PROGRAM P00_OEE
VAR
	//Czasy cyklu 
	fbOEECycleTimes							: FB_OEECycleTimes;
	//Powody odrzuceń           			
	fbOEERejectionReason1					: FB_OEERejectionReason;
	fbOEERejectionReason2					: FB_OEERejectionReason;
	//Przezbrajanie             			
	fbMachinePartsChangeover				: FB_InputFilter;
	
	rtChangeover							: R_TRIG;
	rtfbOEERejectionReason2bDone			: R_TRIG;
	
	sOEERejectionReason1Temp				: STRING;
	sOEERejectionReason2Temp				: STRING;
	
	ifbOEERejectionReason2bAddReasonCount	: INT;
	ifbOEERejectionReason1bAddReasonCount	: INT;
	irtfbOEERejectionReason2bDoneCount		: INT;
	rtfbOEERejectionReason1bDone: R_TRIG;
	irtfbOEERejectionReason1bDoneCount: INT;
	rtORRAdd1sec: R_TRIG;
	tofIbBottleInFormCheckBottleSensor : TOF;

	fbOEERaportLog							: FB_SaveLineToFile;	
	rtOEERaportLogAddLine					: R_TRIG;
	wOEERaportMinuteTemp					: WORD;

	fbOEERaportRejectionLog					: FB_SaveLineToFile;	
	sOEEDateAndTime							: STRING;
	sOEEFileDateAndTime						: STRING;
	sOEEFRejectionLine						: STRING;
	rtOEERaportChooseRecipe					: R_TRIG;	
	bOEETest1								: BOOL;
	tonbOEEGenRaport						: TON;
	sOEEActiveErrorIDs						: STRING;
END_VAR

aCycleTimes();
aRejectionReason();
aMachinePartsChangeover();
aOEETime();
aOEERaport();
aOEEPackMLSuspendedReason();

ACTION aCycleTimes:


tMachineCycleTime;

P02_Dispencers.fbDispencersDragRightStation.tCycleTime;
P02_Dispencers.fbDispencersDragLeftStation.tCycleTime;

P02_Dispencers.fbDispencer1.tCycleTime;
P02_Dispencers.fbDispencer2.tCycleTime;
P02_Dispencers.fbDispencer3.tCycleTime;
P02_Dispencers.fbDispencer4.tCycleTime;
P02_Dispencers.fbDispencerGatesStation.tCycleTime;
P02_Dispencers.fbDispencersCatch1Station.tCycleTime;
P02_Dispencers.fbDispencersCatch2Station.tCycleTime;
P02_Dispencers.fbDispencersCatch3Station.tCycleTime;
P02_Dispencers.fbDispencersCatch4Station.tCycleTime;


P05_Weight.fbWeight1.tCycleTime;
P05_Weight.fbWeight2.tCycleTime;
P05_Weight.fbWeight3.tCycleTime;
P05_Weight.fbWeight4.tCycleTime;


P09_CapPuttedCheck.fbCapPuttedCheck.tCycleTime;

P10_GripperScrewer.fb2GripperScrewer1.tCycleTime;
P10_GripperScrewer.fb2GripperScrewer2.tCycleTime;
P10_GripperScrewer.fbGripperScrewer1CatchStation.tCycleTime;
P10_GripperScrewer.fbGripperScrewer2CatchStation.tCycleTime;

P01_Gates.fbGateBeforeDispencers.tCycleTime;
P13_BottleTransfer.fbBottleTransfer.tCycleTime;




fbOEECycleTimes(
	bEnable:= TRUE, 
	bReset:= FALSE, 
	tStation1CT:= tMachineCycleTime, 
	bStation1En:= TRUE, 
	sStation1Name:= 'M', 
	tStation2CT:= P01_BottleFeeder.fbBottleFeeder.tCycleTime, 
	bStation2En:= P01_BottleFeeder.fbBottleFeeder.bEnable, 
	sStation2Name:= 'SORB', 
	tStation3CT:= P02_Dispencers.fbDispencersDragRightStation.tCycleTime , 
	bStation3En:= P02_Dispencers.fbDispencersDragRightStation.bEnable, 
	sStation3Name:= 'PFDP', 
	tStation4CT:= P02_Dispencers.fbDispencersDragLeftStation.tCycleTime, 
	bStation4En:= P02_Dispencers.fbDispencersDragLeftStation.bEnable, 
	sStation4Name:= 'PFDL', 
	tStation5CT:= P02_Dispencers.fbDispencer1.tCycleTime, 
	bStation5En:= P02_Dispencers.fbDispencer1.bEnable, 
	sStation5Name:= 'D1', 
	tStation6CT:= P02_Dispencers.fbDispencer2.tCycleTime, 
	bStation6En:= P02_Dispencers.fbDispencer2.bEnable,
	sStation6Name:= 'D2', 
	tStation7CT:= P02_Dispencers.fbDispencer3.tCycleTime, 
	bStation7En:= P02_Dispencers.fbDispencer3.bEnable, 
	sStation7Name:= 'D3', 
	tStation8CT:= P02_Dispencers.fbDispencer4.tCycleTime, 
	bStation8En:= P02_Dispencers.fbDispencer4.bEnable, 
	sStation8Name:= 'D4', 
	tStation9CT:= P02_Dispencers.fbDispencersCatch1Station.tCycleTime,
	bStation9En:= P02_Dispencers.fbDispencersCatch1Station.bEnable, 
	sStation9Name:= 'CHD1', 
	tStation10CT:= P02_Dispencers.fbDispencersCatch2Station.tCycleTime, 
	bStation10En:= P02_Dispencers.fbDispencersCatch2Station.bEnable, 
	sStation10Name:= 'CHD2', 
	tStation11CT:= P02_Dispencers.fbDispencersCatch3Station.tCycleTime, 
	bStation11En:= P02_Dispencers.fbDispencersCatch3Station.bEnable,
	sStation11Name:= 'CHD3', 
	tStation12CT:=  P02_Dispencers.fbDispencersCatch4Station.tCycleTime, 
	bStation12En:= P02_Dispencers.fbDispencersCatch4Station.bEnable, 
	sStation12Name:=  'CHD4', 
	tStation13CT:= P05_Weight.fbWeightStation.tCycleTime,
	bStation13En:= P05_Weight.fbWeightStation.bEnable, 
	sStation13Name:= 'PW',
	tStation14CT:= P05_Weight.fbWeightStation2Phase.tCycleTime,
	bStation14En:= P05_Weight.fbWeightStation2Phase.bEnable, 
	sStation14Name:= 'PW',	
	tStation15CT:= P05_Weight.fbWeight1.tCycleTime, 
	bStation15En:= P05_Weight.fbWeight1.bEnable, 
	sStation15Name:= 'W1', 
	tStation16CT:= P05_Weight.fbWeight2.tCycleTime, 
	bStation16En:= P05_Weight.fbWeight2.bEnable, 
	sStation16Name:= 'W2',  
	tStation17CT:= P05_Weight.fbWeight3.tCycleTime, 
	bStation17En:= P05_Weight.fbWeight3.bEnable, 
	sStation17Name:= 'W3',  
	tStation18CT:= P05_Weight.fbWeight4.tCycleTime, 
	bStation18En:= P05_Weight.fbWeight4.bEnable, 
	sStation18Name:= 'W4',  
	tStation19CT:= P05_Weight.fbWeight5.tCycleTime,  
	bStation19En:= P05_Weight.fbWeight5.bEnable,
	sStation19Name:= 'W5',
	tStation20CT:= P05_Weight.fbWeight6.tCycleTime,  
	bStation20En:= P05_Weight.fbWeight6.bEnable, 
	sStation20Name:= 'W6',  
	tStation21CT:= P10_GripperScrewer.fbGripperScrewersDragStation.tCycleTime, 
	bStation21En:= P10_GripperScrewer.fbGripperScrewersDragStation.bEnable,
	sStation21Name:= 'PFDZ',
	tStation22CT:= P10_GripperScrewer.fb2GripperScrewer1.tCycleTime, 
	bStation22En:= P10_GripperScrewer.fb2GripperScrewer1.bEnable1,
	sStation22Name:= 'ZS1',
	tStation23CT:= P10_GripperScrewer.fb2GripperScrewer2.tCycleTime, 
	bStation23En:= P10_GripperScrewer.fb2GripperScrewer2.bEnable2,
	sStation23Name:= 'ZS2',
	tStation24CT:= P10_GripperScrewer.fbGripperScrewersDragStation.tCycleTime, 
	bStation24En:= P10_GripperScrewer.fbGripperScrewersDragStation.bEnable,
	sStation24Name:= 'PFZ',
	tStation25CT:= P10_GripperScrewer.fbGripperScrewer1CatchStation.tCycleTime, 
	bStation25En:= P10_GripperScrewer.fbGripperScrewer1CatchStation.bEnable,
	sStation25Name:= 'CHZS1',
	tStation26CT:= P10_GripperScrewer.fbGripperScrewer2CatchStation.tCycleTime, 
	bStation26En:= P10_GripperScrewer.fbGripperScrewer2CatchStation.bEnable,
	sStation26Name:= 'CHZS2',
	tStation27CT:= P11_CapCorrectCheck.fbCapCorrectCheck.tCycleTime, 
	bStation27En:= P11_CapCorrectCheck.fbCapCorrectCheck.bEnable,
	sStation27Name:= 'SZA',
	tStation28CT:= P13_BottleTransfer.fbBottleTransfer.tCycleTime, 
	bStation28En:= P13_BottleTransfer.fbBottleTransfer.bEnable,
	sStation28Name:= 'R',  
	tStation29CT:= P01_Gates.fbGateBeforeDispencers.tCycleTime, 
	bStation29En:= P01_Gates.fbGateBeforeDispencers.bEnable, 
	sStation29Name:= 'SZD', 
	tStation20CT:= P01_Gates.fbGateRobot.tCycleTime, 
	bStation30En:= P01_Gates.fbGateRobot.bEnable, 
	sStation30Name:= 'SZR', 

	
	
	AsCycleTimes=> VIS.AsOEECycleTimes,
	
	
	
	);
END_ACTION

ACTION aMachinePartsChangeover:

VIS.bMachinePartsChangeOver	;						// Włączone przezbrajanie (ustawić z wizki)
VIS.iMachinePartsChangeOver	;						// Stan przezbrajania (0-ruch,1-pozycja gorna,-1-pozycja dolna) 
VIS.bBottleSorterDisable	;						// Wyłączenie sortera butelek
VIS.bCapSorterDisable		;						// Wyłączenie sortera nasadek


//Sygnał z wizki
VIS.bMachinePartsChangeover;
//Filtrowanie sygnału, przeciw lagom z wizualizacji lub ciągłym klikaniem
fbMachinePartsChangeover(bIn:=VIS.bMachinePartsChangeover,tFilterTimeOn:=T#3S,tFilterTimeOff:=T#3S,bOUT=>bChangeover);
//Przefiltrowany
bChangeover;

VIS.iMachinePartsChangeOver;
// Trzeba dodać, albo wyłączona stacja!
//Przezbrajanie - okienko 


IF bChangeover THEN
	VIS.bBottleSorterHold	:= TRUE;	
	VIS.bCapSorterHold		:= TRUE;	
	//VIS.bTank1SupplyPumpEnableShow:=FALSE;
	//VIS.bTank2SupplyPumpEnableShow:=FALSE;
ELSE
	//VIS.bBottleSorterHold	:= FALSE;	
	VIS.bCapSorterHold		:= FALSE;			
END_IF

IF 
 (P02_Dispencers.fbDispencersCatch1Station.eState = E_Station.ePreparingToDisable 			OR P02_Dispencers.fbDispencersCatch1Station.eState = E_Station.eHoming 				OR (NOT bDispencer1Enable AND NOT bDispencer3Enable)) 																			AND
 (P09_CapPuttedCheck.fbCapPuttedCheck.eState = E_Station.ePreparingToDisable				OR P09_CapPuttedCheck.fbCapPuttedCheck.eState = E_Station.eHoming				 	OR NOT bCapPuttedCheckEnable) 									AND
 (P10_GripperScrewer.fb2GripperScrewer1.eState = E_Station.ePreparingToDisable				OR P10_GripperScrewer.fb2GripperScrewer1.eState = E_Station.eHoming  				OR NOT bGripperScrewer1Enable) 									AND
 (P10_GripperScrewer.fb2GripperScrewer2.eState = E_Station.ePreparingToDisable				OR P10_GripperScrewer.fb2GripperScrewer2.eState = E_Station.eHoming  				OR NOT bGripperScrewer2Enable)									AND
 (P10_GripperScrewer.fbGripperScrewer1CatchStation.eState = E_Station.ePreparingToDisable 	OR P10_GripperScrewer.fbGripperScrewer1CatchStation.eState = E_Station.eHoming		OR NOT bGripperScrewer1Enable) 									AND
 (P10_GripperScrewer.fbGripperScrewer2CatchStation.eState = E_Station.ePreparingToDisable 	OR P10_GripperScrewer.fbGripperScrewer2CatchStation.eState = E_Station.eHoming 		OR NOT bGripperScrewer2Enable) 									AND
 (P11_CapCorrectCheck.fbCapCorrectCheck.eState = E_Station.ePreparingToDisable 				OR P11_CapCorrectCheck.fbCapCorrectCheck.eState = E_Station.eHoming					OR NOT bCapCorrectCheckEnable)
THEN
    VIS.iMachinePartsChangeOver := 0; //ruch
ELSIF
  (P02_Dispencers.fbDispencersCatch1Station.eState = E_Station.eDisabled			OR P02_Dispencers.fbDispencersCatch1Station.eState = E_Station.eManualMovement 			OR (NOT bDispencer1Enable AND NOT bDispencer3Enable) ) 											AND
 (P09_CapPuttedCheck.fbCapPuttedCheck.eState = E_Station.eDisabled				 	OR NOT bCapPuttedCheckEnable) 										AND
 (P10_GripperScrewer.fb2GripperScrewer1.eState = E_Station.eDisabled  				OR NOT bGripperScrewer1Enable)										AND
 (P10_GripperScrewer.fb2GripperScrewer2.eState = E_Station.eDisabled  				OR	NOT bGripperScrewer2Enable)										AND
 (P10_GripperScrewer.fbGripperScrewer1CatchStation.eState = E_Station.eDisabled 	OR NOT bGripperScrewer1Enable) 										AND
 (P10_GripperScrewer.fbGripperScrewer2CatchStation.eState = E_Station.eDisabled 	OR NOT bGripperScrewer2Enable) 										AND
 (P11_CapCorrectCheck.fbCapCorrectCheck.eState = E_Station.eDisabled 				OR NOT bCapCorrectCheckEnable)
THEN
    VIS.iMachinePartsChangeOver := 1; //1 pozycja gorna
ELSIF 
  (P02_Dispencers.fbDispencersCatch1Station.eState = E_Station.eReady 		OR P02_Dispencers.fbDispencersCatch1Station.eState = E_Station.eManualMovement 				OR (NOT bDispencer1Enable AND NOT bDispencer3Enable)) 												AND
 (P09_CapPuttedCheck.fbCapPuttedCheck.eState = E_Station.eReady				OR P09_CapPuttedCheck.fbCapPuttedCheck.eState = E_Station.eManualMovement			 		OR NOT bCapPuttedCheckEnable) 											AND
 (P10_GripperScrewer.fb2GripperScrewer1.eState = E_Station.eReady  			OR P10_GripperScrewer.fb2GripperScrewer1.eState = E_Station.eManualMovement					OR NOT bGripperScrewer1Enable)											AND
 (P10_GripperScrewer.fb2GripperScrewer2.eState = E_Station.eReady  			OR P10_GripperScrewer.fb2GripperScrewer2.eState = E_Station.eManualMovement					OR NOT bGripperScrewer2Enable) 											AND
 (P10_GripperScrewer.fbGripperScrewer1CatchStation.eState = E_Station.eReady OR P10_GripperScrewer.fbGripperScrewer1CatchStation.eState = E_Station.eManualMovement		OR NOT bGripperScrewer1Enable) 											AND
 (P10_GripperScrewer.fbGripperScrewer2CatchStation.eState = E_Station.eReady OR P10_GripperScrewer.fbGripperScrewer2CatchStation.eState = E_Station.eManualMovement		OR NOT bGripperScrewer2Enable) 											AND
 (P11_CapCorrectCheck.fbCapCorrectCheck.eState = E_Station.eReady 			OR	P11_CapCorrectCheck.fbCapCorrectCheck.eState = E_Station.eManualMovement 				OR NOT bCapCorrectCheckEnable)
THEN
    VIS.iMachinePartsChangeOver := -1; // -1pozycja dolna
END_IF 

//Kasowanie cyklu i liczników
rtChangeover(CLK:=bChangeover,Q=>);
IF rtChangeover.Q THEN
	//bCycleReseting := TRUE;	
	VIS.uiCounterAverageEfficiency:=0;
	VIS.udiCounterShiftBottles:=0;
	VIS.uiCounterInstantEfficiency:=0;
	VIS.uiCounterGoodBottles:=0;
	VIS.uiCounterBadBottles:=0;
END_IF
END_ACTION

ACTION aOEEPackMLSuspendedReason:
(*
Nazwa:			aOEEPackMLSuspendedReason
Wersja:			v0.1 			
Autor:			DP
Urzadzenia:		HMI, 
Konfiguracja:	
Info:
- Wyświetlanie na wykresie powodu zatrzymania lini, czyli w przyszłości przjeścia w stan PackML ->Suspended
Uwagi:

Zmiany:

*)
IF P00_PackML.tonCycleBadBottleConveyorFullSensor.Q THEN //odrzut
	VIS.iOEEPackMLSuspendedReason	:= 1;
ELSIF P16_LabelMachine.tonLabelMachineFullSensorInfo.Q THEN 
	//IF VIS.UPPackMLState=6 AND VIS.EPPackMLState=6 THEN		//etykieciarka
	VIS.iOEEPackMLSuspendedReason	:= 2;
ELSIF	vis.iMachineState = 2 OR vis.iMachineState = 8 OR vis.iMachineState = 9 OR vis.iMachineState = 15 THEN
	VIS.iOEEPackMLSuspendedReason	:= 3;
	//ELSIF VIS.UPPackMLState<>6 AND VIS.EPPackMLState=6 THEN //kartoniarka
	//VIS.iOEEPackMLSuspendedReason	:= 7;
	//ELSIF VIS.UPPackMLState=6 AND VIS.EPPackMLState<>6 THEN //paletyzer
	//VIS.iOEEPackMLSuspendedReason	:= 8;
	//END_IF
//ELSIF VIS.uliWarningOccure.33 THEN  //brak butelek
//	VIS.iOEEPackMLSuspendedReason	:= 3;	
//ELSIF VIS.uliWarningOccure.27 THEN	//brak nakrętek
//	VIS.iOEEPackMLSuspendedReason	:= 4;	
//(*ELSIF NOT P16_LabelMachine.tonLabelMachineFullSensorInfo.Q THEN		
//	IF VIS.UPPackMLState<>6 AND VIS.EPPackMLState=6 THEN			//kartoniarka
//	VIS.iOEEPackMLSuspendedReason	:= 7;
//	ELSIF VIS.UPPackMLState=6 AND VIS.EPPackMLState<>6 THEN			//paletyzer
//	VIS.iOEEPackMLSuspendedReason	:= 8;
//	END_IF*)
ELSE
	VIS.iOEEPackMLSuspendedReason	:= 0;		
END_IF
END_ACTION

ACTION aOEERaport:

//Data dla danych - według opisu
sOEEDateAndTime:= 
Concat(Concat(Concat(Concat(Concat(Concat(Concat(Concat(Concat(Concat(Concat(WORD_TO_STRING(wDay),'.'),WORD_TO_STRING(wMonth)),'.'),WORD_TO_STRING(wYear)),';'),WORD_TO_STRING(wHour)),':'),WORD_TO_STRING(wMinute)),';'),''),'');

//Generowanie raportu z wizki - podpiąć pod wybór receptury?
VIS.bOEEGenRaport;

//Zapisywanie daty wybrania receptury
//rtOEERaportChooseRecipe(CLK:=VIS.bChooseRecipe OR bOEETest1, Q=>);
rtOEERaportChooseRecipe(CLK:=VIS.bOEEGenRaport OR bOEETest1, Q=>);
tonbOEEGenRaport(IN:=VIS.bOEEGenRaport, PT:=T#500MS);
IF rtOEERaportChooseRecipe.Q THEN
	sOEEFileDateAndTime:= 
	Concat(Concat(Concat(Concat(Concat(Concat(Concat(Concat(Concat(Concat(Concat(WORD_TO_STRING(wYear),''),WORD_TO_STRING(wMonth)),''),WORD_TO_STRING(wDay)),''),WORD_TO_STRING(wHour)),''),WORD_TO_STRING(wMinute)),''),''),'');
	bOEETest1	:=	FALSE;
END_IF
IF tonbOEEGenRaport.Q THEN
	VIS.bOEEGenRaport	:= FALSE;
END_IF

//Zapisywanie danych co 1 min
rtOEERaportLogAddLine(CLK:=wMinute <> wOEERaportMinuteTemp, Q=>);	
IF rtOEERaportLogAddLine.Q THEN 
	wOEERaportMinuteTemp := wMinute;
END_IF

//Zapisywanie aktywnych bledow w stringu
IF rtOEERaportLogAddLine.Q THEN
	sOEEActiveErrorIDs := '';
	FOR i:=1 TO 10 DO
		IF VIS.fbAlarms.arrActiveEvents[i].stEventEntry.nEventId <> 0 THEN
			sOEEActiveErrorIDs:=Concat(sOEEActiveErrorIDs,Concat(UDINT_TO_STRING(VIS.fbAlarms.arrActiveEvents[i].stEventEntry.nEventId),';'));	
		END_IF
	END_FOR
	sOEEActiveErrorIDs:= Concat(sOEEActiveErrorIDs,stBottleSorterRead.eError.sStationName);
	sOEEActiveErrorIDs:= Concat(sOEEActiveErrorIDs,stCapSorterRead.eError.sStationName);	
END_IF			
		
//Raport nazwy,liczników itd
fbOEERaportLog(
	bExecute:= rtOEERaportLogAddLine.Q,
	AmsNetId:= , 
	sPath:='C:\Users\Administrator\Desktop\CSVFolder\', 
	sName:= Concat(sOEEFileDateAndTime,	Concat('-',Concat(sRecipeName,'.csv'))), 
	sLine:= 
	
Concat(
	'$R$N',
	Concat(
		sOEEDateAndTime,
		Concat(
				UINT_TO_STRING(VIS.iMachineState),
				Concat(
						';',
							Concat(
									sRecipeName,
									Concat(
											';',
											Concat(
													UDINT_TO_STRING(VIS.udiCounterGlobal),
														Concat(
																';',
																	Concat(
																		UDINT_TO_STRING(VIS.uiCounterBadBottles),
																		Concat(
																			';',
																			Concat(
																					//UDINT_TO_STRING(VIS.udiStationErrorCode),
																					sOEEActiveErrorIDs,
																					';'
																					)	
																				)	
																			)
																)
													)
											)
										)
						)
					)
				)
		)		
	,
	
	bBusy=>, 
	bError=>);

	IF rtOEERaportLogAddLine.Q THEN
		sOEEFRejectionLine := '';
		FOR i:= 0 TO 63 DO
			IF 	VIS.AStBadPackageReason[i].udiID <> 0 THEN
				
				sOEEFRejectionLine := 
					Concat(sOEEFRejectionLine,Concat(UDINT_TO_STRING(VIS.AStBadPackageReason[i].udiID), Concat(';',Concat(WSTRING_TO_STRING(VIS.AStBadPackageReason[i].wsDescription),';'))));
						
			END_IF
		END_FOR
	END_IF

//Raport odrzutów
fbOEERaportRejectionLog(
	bExecute:= rtOEERaportLogAddLine.Q,
	AmsNetId:= , 
	sPath:='C:\Users\Administrator\Desktop\CSVRejectionFolder\', 
	sName:= Concat(sOEEFileDateAndTime,	Concat('-',Concat(sRecipeName,'-Rejection.csv'))), 
	sLine:= Concat('$R$N',sOEEFRejectionLine),
	bBusy=>, 
	bError=>);
END_ACTION

ACTION aOEETime:

VIS.udiCounterShiftBottles;
VIS.udiCounterGlobal;            
VIS.udiCounterGlobalBadBottles;     

VIS.sOEEText1 := Concat(Concat('PRACA: ', UDINT_TO_STRING(udiCounterExecuteTimeTemp/60)),' min');
VIS.sOEEText2 := Concat(Concat('POSTÓJ: ', UDINT_TO_STRING(udiCounterReadyTimeTemp/60)),' min');
VIS.sOEEText3 := Concat(Concat('BŁĄD: ', UDINT_TO_STRING(udiCounterErrorTimeTemp/60)),' min');
tofIbBottleInFormCheckBottleSensor(IN:=MAIN.IbBottleInFormCheckBottleSensor,PT:=T#30S);

VIS.udiCounterExecuteTime	:=	UDINT_TO_UINT(udiCounterExecuteTimeTemp/60);
VIS.udiCounterReadyTime		:=	UDINT_TO_UINT(udiCounterReadyTimeTemp/60);
VIS.udiCounterErrorTime	  	:=	UDINT_TO_UINT(udiCounterErrorTimeTemp/60);
rtORRAdd1sec(CLK:=b2Hz,Q=>);

IF	
	//P00_PackML.fbPMLAuto.ePMLState = Tc3_PackML.E_PMLState.ePMLState_STARTING OR 
	//P00_PackML.fbPMLAuto.ePMLState = Tc3_PackML.E_PMLState.ePMLState_STOPPING OR 
	P00_PackML.fbPMLAuto.ePMLState = Tc3_PackML.E_PMLState.ePMLState_EXECUTE AND
	tofIbBottleInFormCheckBottleSensor.Q AND 
	NOT P16_LabelMachine.tonLabelMachineFullSensorInfo.Q AND
	NOT (P00_PackML.tonCycleBadBottleConveyorFullSensor.Q AND (P00_PackML.iRobotPickCase=110 OR P00_PackML.iRobotPickCase=210))
	THEN

	IF rtORRAdd1sec.Q THEN
		udiCounterExecuteTimeTemp	:=	udiCounterExecuteTimeTemp	+	1;
		
	END_IF
	
ELSIF
	P00_PackML.fbPMLAuto.ePMLState = Tc3_PackML.E_PMLState.ePMLState_STOPPED OR 
	P00_PackML.fbPMLAuto.ePMLState = Tc3_PackML.E_PMLState.ePMLState_ABORTED  
	THEN
	
	IF rtORRAdd1sec.Q THEN
		udiCounterErrorTimeTemp	:=	udiCounterErrorTimeTemp	+	1;
	END_IF	

ELSE
	IF rtORRAdd1sec.Q THEN
		udiCounterReadyTimeTemp	:=	udiCounterReadyTimeTemp	+	1;
	END_IF	
END_IF
END_ACTION

ACTION aRejectionReason:

//może uzależnić też od ilości opakowań do pobrania VIS.nBottleTransferPickOption			:=	1; // 1 butelka
//													VIS.nBottleTransferPlaceOption			:=	2; //Odrzucone butelki 

fbOEERejectionReason1(
                        bEnable				:= TRUE,
                        bReset				:= ,
                        udiGlobalCounter	:= VIS.udiCounterGlobal, //Globalny licznik konfekcji [szt]
                        bAddReason			:= P13_BottleTransfer.fbBottleTransfer.eRunningState>1 AND VIS.nBottleTransferPlaceOption=2, // może dodać dodatkowy warunek?
                        bReason1			:= eRobotPackageState[1].bWeightTooLow 			AND eRobotPackageState[1].bBottlePresent,
                        sReason1Description	:= 'WZM',
                        bReason2			:= eRobotPackageState[1].bWeightTooHigh 		AND eRobotPackageState[1].bBottlePresent,
                        sReason2Description	:= 'WZD',
                        bReason3			:= NOT eRobotPackageState[1].bCapOK 			AND eRobotPackageState[1].bBottlePresent,
                        sReason3Description	:= 'BNPZ',
                        bReason4			:= NOT eRobotPackageState[1].bCapGripperScrewed AND eRobotPackageState[1].bBottlePresent,
                        sReason4Description	:= 'NZZSZ',
                        bReason5			:= NOT eRobotPackageState[1].bCapCorrectCapOn 	AND eRobotPackageState[1].bBottlePresent,
                        sReason5Description	:= 'BNZZ',
                        bReason6			:= eRobotPackageState[1].bCapCorrectNOK 		AND eRobotPackageState[1].bBottlePresent,
                        sReason6Description	:= 'NZZ',
                        bReason7			:=, 
                        sReason7Description	:= ,      
                        sRejectionReason	:= sOEERejectionReason1Temp,
                        );

fbOEERejectionReason2(
                        bEnable				:= TRUE,
                        bReset				:= ,
                        udiGlobalCounter	:= VIS.udiCounterGlobal, //Globalny licznik konfekcji [szt]
                        bAddReason			:= P13_BottleTransfer.fbBottleTransfer.eRunningState>1 AND VIS.nBottleTransferPlaceOption=2,
                        bReason1			:= eRobotPackageState[2].bWeightTooLow 			AND eRobotPackageState[2].bBottlePresent,
                        sReason1Description	:= 'WZM',
                        bReason2			:= eRobotPackageState[2].bWeightTooHigh 		AND eRobotPackageState[2].bBottlePresent,
                        sReason2Description	:= 'WZD',
                        bReason3			:= NOT eRobotPackageState[2].bCapOK 			AND eRobotPackageState[2].bBottlePresent,
                        sReason3Description	:= 'BNPZ',
                        bReason4			:= NOT eRobotPackageState[2].bCapGripperScrewed AND eRobotPackageState[2].bBottlePresent,
                        sReason4Description	:= 'NZZSZ',
                        bReason5			:= NOT eRobotPackageState[2].bCapCorrectCapOn 	AND eRobotPackageState[2].bBottlePresent,
                        sReason5Description	:= 'BNZZ',
                        bReason6			:= eRobotPackageState[2].bCapCorrectNOK 		AND eRobotPackageState[2].bBottlePresent,
                        sReason6Description	:= 'NZZ',
                        bReason7			:= , 
                        sReason7Description	:= ,      
                        sRejectionReason	:= sOEERejectionReason2Temp,
                        );
						
	rtfbOEERejectionReason2bDone(CLK:=fbOEERejectionReason2.bDone,Q=>);
	rtfbOEERejectionReason1bDone(CLK:=fbOEERejectionReason1.bDone,Q=>);
// dodałem na testy! 20.06	
	IF rtfbOEERejectionReason1bDone.Q AND  VIS.nBottleTransferPickOption=1 THEN
		VIS.sOEERejectionReason 			:=sOEERejectionReason1Temp;//	CONCAT(sOEERejectionReason1Temp,';');
		irtfbOEERejectionReason1bDoneCount	:=	irtfbOEERejectionReason1bDoneCount+1;
	END_IF
	
	
	IF rtfbOEERejectionReason2bDone.Q AND  VIS.nBottleTransferPickOption=2 THEN
		VIS.sOEERejectionReason 			:=	CONCAT(CONCAT(sOEERejectionReason1Temp,';'),sOEERejectionReason2Temp);
		irtfbOEERejectionReason2bDoneCount	:=	irtfbOEERejectionReason2bDoneCount+1;
	END_IF
	
    //Przeniesione dodawanie liczników, po to żeby dla wizualizacji i skryptów było łatwiej (kolejnosć odczytu)
    IF bAddGlobalCounter AND (fbOEERejectionReason2.bDone OR fbOEERejectionReason1.bDone )THEN
        VIS.uiCounterBadBottles                	:= VIS.uiCounterBadBottles		+ INT_TO_UINT(P00_PackML.nCounterFormsToLoad);//+ 1;// czy aby na pewno +1 ???
        VIS.udiCounterGlobalBadBottles        	:= VIS.udiCounterGlobalBadBottles	+ INT_TO_UDINT(P00_PackML.nCounterFormsToLoad);
        VIS.udiCounterGlobal                   	:= VIS.udiCounterGlobal			+ INT_TO_UDINT(P00_PackML.nCounterFormsToLoad);
        //VIS.udiCounterShiftBottles            	:= VIS.udiCounterShiftBottles	+ INT_TO_UDINT(P00_PackML.nCounterFormsToLoad);
        bAddGlobalCounter                    	:= FALSE;
    END_IF

    IF fbOEERejectionReason1.bAddReason THEN
       ifbOEERejectionReason1bAddReasonCount:=ifbOEERejectionReason1bAddReasonCount+1;
    END_IF
	
    IF fbOEERejectionReason2.bAddReason THEN
        ifbOEERejectionReason2bAddReasonCount:=ifbOEERejectionReason2bAddReasonCount+1;
     END_IF
END_ACTION

END_PROGRAM

(* stored: Version 1.1.0.1, ProductVersion 3.1.4026.13, FileIdentifier 02689428d8efeed8a78b8ef3a3fdcfe5d09039a9, FileSignature 44daf26e7e7288f74d3f978d1d0214b2b1e5c506aa9bfd24740d0514adf3d7f1fed84f6822c00263c792253789ebda25bdc56938ff42e3c47365d65a564f3c8034953b4d2f9a46ca5952431417d125fd436c812405c40c2e3f75dcfe042a473413b156317058a588511bcd444fc63c9d2a5edcfb8a3e4d1b3007ca2dd304362b15f63a3ef2c8624fa66b21e5af4a2dada87096a7028e7d86cdc7e0a1abc17373387c7f25656e002f963e77048528c9d3ee5a8664849fcff38f7fdd1dda37988d09f68298b31ae6fe10a5b95e2b73eac28d16b4fce65a3f435e9996781ee949c42ed40e4418f2cb3d264bd489d0da85916129245d2c4672d1935a82bfee9b4390
   POU P00_OEE: Id {08c14e30-ec5a-4e4c-b5ac-ce8b40bd55d7}, SpecialFunc None
   Action aCycleTimes: Id {31f9078a-cb7d-46d4-a01e-ed62c78a0b70}
   Action aMachinePartsChangeover: Id {d8efbd55-9884-473e-b9ad-c53d3aedee1b}
   Action aOEEPackMLSuspendedReason: Id {0f2ca1c6-2b3d-4dcc-8e48-a41de4d60df8}
   Action aOEERaport: Id {eb349611-227d-4b80-8b71-60ce228f0e50}
   Action aOEETime: Id {68dc93d9-107e-4735-be6d-99896abcd4f7}
   Action aRejectionReason: Id {15f5a4bb-fd9b-4e2f-b048-7aca5d85e754} *)
